Staubli VAL3: CommType.dtx

public num INVALID
public num TOPIC
public num SERVICE_REQUEST
public num SERVICE_REPLY
